PROGRAM F33_OuterPrinters_v2_Evo
VAR
	aSquareWave		 		: ARRAY[1..2] OF  FB_SquareWave;
	aOuterCodeGenerator 		: ARRAY[1..2] OF  FB_CODE_OuterCodeGenerator;
	aSelectCommand	 		: ARRAY[1..2] OF  FB_PRINTER_SelectCommand;

	aLabelPrintCtrl				: ARRAY[1..2] OF  RS;
	aLabelApplyCtrl			: ARRAY[1..2] OF  RS;

	tonLoweratorAtConstSpeed	: TON;
	rsInhibitLabbeller1Apply		: RS	;
	rsInhibitLabbeller2Apply		: RS	;

	fbDebugCNT				: FB_DEBUG_CounterArray;
	aCNTDebug				: ARRAY [1..10] OF UDINT;
	bResetCNT				: BOOL;
	bEnableResendCommand		: BOOL;
	rtEncoder	: R_TRIG;
END_VAR
VAR // added by the converter: edge detectors and wires of the graphical bodies
    _w1, _w2, _w3 : BOOL;
    _w4, _w5, _w6 : ANY;
END_VAR

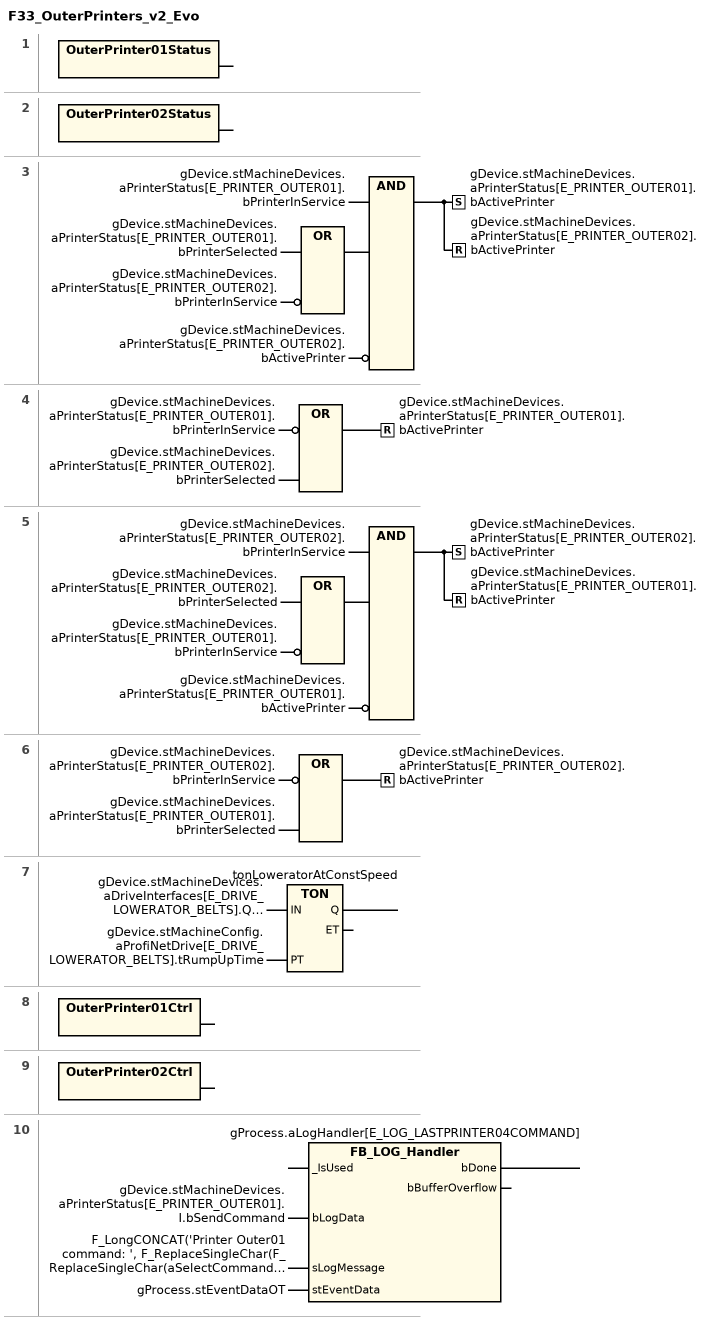
// NETWORK 1
OuterPrinter01Status();

// NETWORK 2
OuterPrinter02Status();

// NETWORK 3
_w1 := gDevice.stMachineDevices.aPrinterStatus[E_PRINTER_OUTER01].bPrinterInService AND (gDevice.stMachineDevices.aPrinterStatus[E_PRINTER_OUTER01].bPrinterSelected OR NOT gDevice.stMachineDevices.aPrinterStatus[E_PRINTER_OUTER02].bPrinterInService) AND NOT gDevice.stMachineDevices.aPrinterStatus[E_PRINTER_OUTER02].bActivePrinter;
gDevice.stMachineDevices.aPrinterStatus[E_PRINTER_OUTER01].bActivePrinter S= _w1;
gDevice.stMachineDevices.aPrinterStatus[E_PRINTER_OUTER02].bActivePrinter R= _w1;

// NETWORK 4
gDevice.stMachineDevices.aPrinterStatus[E_PRINTER_OUTER01].bActivePrinter R= NOT gDevice.stMachineDevices.aPrinterStatus[E_PRINTER_OUTER01].bPrinterInService OR gDevice.stMachineDevices.aPrinterStatus[E_PRINTER_OUTER02].bPrinterSelected;

// NETWORK 5
_w2 := gDevice.stMachineDevices.aPrinterStatus[E_PRINTER_OUTER02].bPrinterInService AND (gDevice.stMachineDevices.aPrinterStatus[E_PRINTER_OUTER02].bPrinterSelected OR NOT gDevice.stMachineDevices.aPrinterStatus[E_PRINTER_OUTER01].bPrinterInService) AND NOT gDevice.stMachineDevices.aPrinterStatus[E_PRINTER_OUTER01].bActivePrinter;
gDevice.stMachineDevices.aPrinterStatus[E_PRINTER_OUTER02].bActivePrinter S= _w2;
gDevice.stMachineDevices.aPrinterStatus[E_PRINTER_OUTER01].bActivePrinter R= _w2;

// NETWORK 6
gDevice.stMachineDevices.aPrinterStatus[E_PRINTER_OUTER02].bActivePrinter R= NOT gDevice.stMachineDevices.aPrinterStatus[E_PRINTER_OUTER02].bPrinterInService OR gDevice.stMachineDevices.aPrinterStatus[E_PRINTER_OUTER01].bPrinterSelected;

// NETWORK 7
tonLoweratorAtConstSpeed(IN := gDevice.stMachineDevices.aDriveInterfaces[E_DRIVE_LOWERATOR_BELTS].Q.xOperationEnable, PT := gDevice.stMachineConfig.aProfiNetDrive[E_DRIVE_LOWERATOR_BELTS].tRumpUpTime); // TON

// NETWORK 8
OuterPrinter01Ctrl();

// NETWORK 9
OuterPrinter02Ctrl();

// NETWORK 10
gProcess.aLogHandler[E_LOG_LASTPRINTER04COMMAND](
    bLogData := gDevice.stMachineDevices.aPrinterStatus[E_PRINTER_OUTER01].I.bSendCommand,
    sLogMessage := F_LongCONCAT('Printer Outer01 command: ', F_ReplaceSingleChar(F_ReplaceSingleChar(aSelectCommand[1].sPrintCommand, '$N', '_' ), '$R', '_')),
    stEventData := gProcess.stEventDataOT); // FB_LOG_Handler

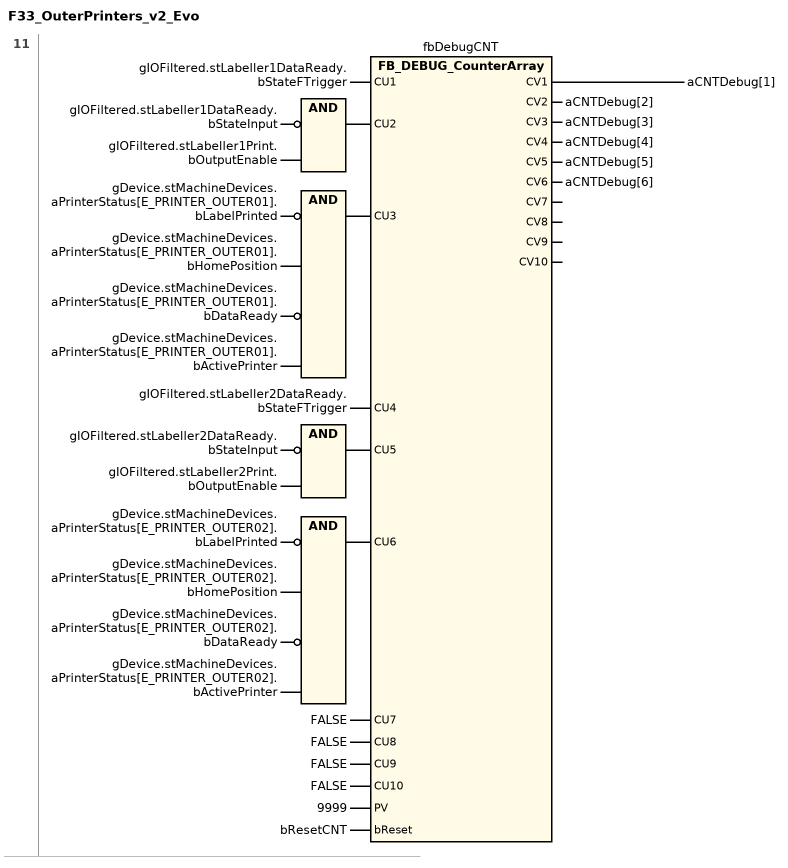
// NETWORK 11
fbDebugCNT(
    CU1 := gIOFiltered.stLabeller1DataReady.bStateFTrigger,
    CU2 := NOT gIOFiltered.stLabeller1DataReady.bStateInput AND gIOFiltered.stLabeller1Print.bOutputEnable,
    CU3 := NOT gDevice.stMachineDevices.aPrinterStatus[E_PRINTER_OUTER01].bLabelPrinted AND gDevice.stMachineDevices.aPrinterStatus[E_PRINTER_OUTER01].bHomePosition AND NOT gDevice.stMachineDevices.aPrinterStatus[E_PRINTER_OUTER01].bDataReady AND gDevice.stMachineDevices.aPrinterStatus[E_PRINTER_OUTER01].bActivePrinter,
    CU4 := gIOFiltered.stLabeller2DataReady.bStateFTrigger,
    CU5 := NOT gIOFiltered.stLabeller2DataReady.bStateInput AND gIOFiltered.stLabeller2Print.bOutputEnable,
    CU6 := NOT gDevice.stMachineDevices.aPrinterStatus[E_PRINTER_OUTER02].bLabelPrinted AND gDevice.stMachineDevices.aPrinterStatus[E_PRINTER_OUTER02].bHomePosition AND NOT gDevice.stMachineDevices.aPrinterStatus[E_PRINTER_OUTER02].bDataReady AND gDevice.stMachineDevices.aPrinterStatus[E_PRINTER_OUTER02].bActivePrinter,
    CU7 := FALSE,
    CU8 := FALSE,
    CU9 := FALSE,
    CU10 := FALSE,
    PV := 9999,
    bReset := bResetCNT,
    CV2 => aCNTDebug[2],
    CV3 => aCNTDebug[3],
    CV4 => aCNTDebug[4],
    CV5 => aCNTDebug[5],
    CV6 => aCNTDebug[6]); // FB_DEBUG_CounterArray
aCNTDebug[1] := fbDebugCNT.CV1;

ACTION OuterPrinter01Ctrl:
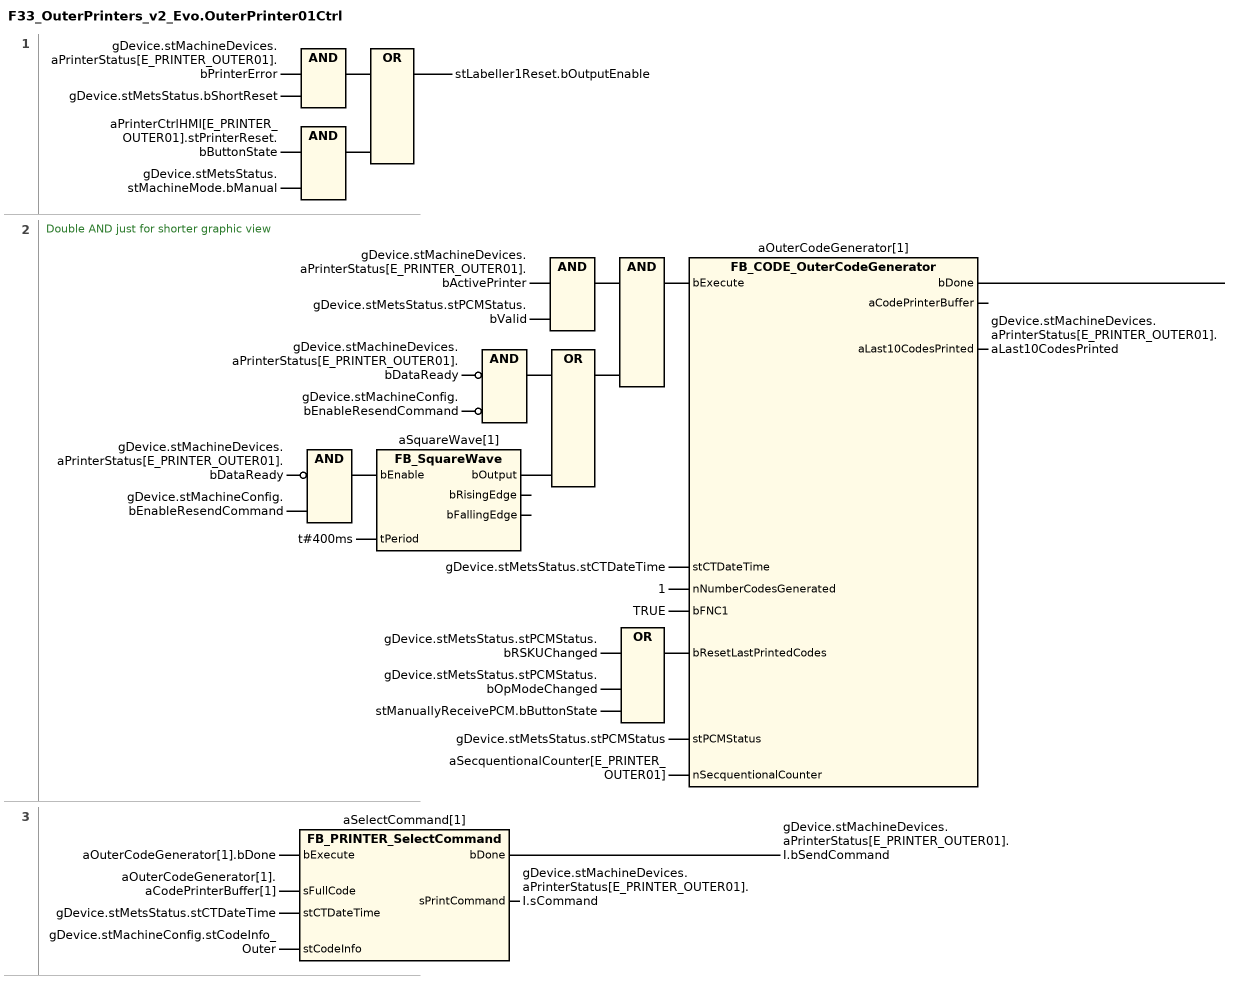
// NETWORK 1
stLabeller1Reset.bOutputEnable := gDevice.stMachineDevices.aPrinterStatus[E_PRINTER_OUTER01].bPrinterError AND gDevice.stMetsStatus.bShortReset OR aPrinterCtrlHMI[E_PRINTER_OUTER01].stPrinterReset.bButtonState AND gDevice.stMetsStatus.stMachineMode.bManual;

// NETWORK 2
// Double AND just for shorter graphic view
aSquareWave[1](bEnable := NOT gDevice.stMachineDevices.aPrinterStatus[E_PRINTER_OUTER01].bDataReady AND gDevice.stMachineConfig.bEnableResendCommand, tPeriod := t#400ms); // FB_SquareWave
aOuterCodeGenerator[1](
    bExecute := (gDevice.stMachineDevices.aPrinterStatus[E_PRINTER_OUTER01].bActivePrinter AND gDevice.stMetsStatus.stPCMStatus.bValid) AND (NOT gDevice.stMachineDevices.aPrinterStatus[E_PRINTER_OUTER01].bDataReady AND NOT gDevice.stMachineConfig.bEnableResendCommand OR aSquareWave[1].bOutput),
    stCTDateTime := gDevice.stMetsStatus.stCTDateTime,
    nNumberCodesGenerated := 1,
    bFNC1 := TRUE,
    bResetLastPrintedCodes := gDevice.stMetsStatus.stPCMStatus.bRSKUChanged OR gDevice.stMetsStatus.stPCMStatus.bOpModeChanged OR stManuallyReceivePCM.bButtonState,
    stPCMStatus := gDevice.stMetsStatus.stPCMStatus,
    nSecquentionalCounter := aSecquentionalCounter[E_PRINTER_OUTER01],
    aLast10CodesPrinted => gDevice.stMachineDevices.aPrinterStatus[E_PRINTER_OUTER01].aLast10CodesPrinted); // FB_CODE_OuterCodeGenerator

// NETWORK 3
aSelectCommand[1](
    bExecute := aOuterCodeGenerator[1].bDone,
    sFullCode := aOuterCodeGenerator[1].aCodePrinterBuffer[1],
    stCTDateTime := gDevice.stMetsStatus.stCTDateTime,
    stCodeInfo := gDevice.stMachineConfig.stCodeInfo_Outer,
    sPrintCommand => gDevice.stMachineDevices.aPrinterStatus[E_PRINTER_OUTER01].I.sCommand); // FB_PRINTER_SelectCommand
gDevice.stMachineDevices.aPrinterStatus[E_PRINTER_OUTER01].I.bSendCommand := aSelectCommand[1].bDone;

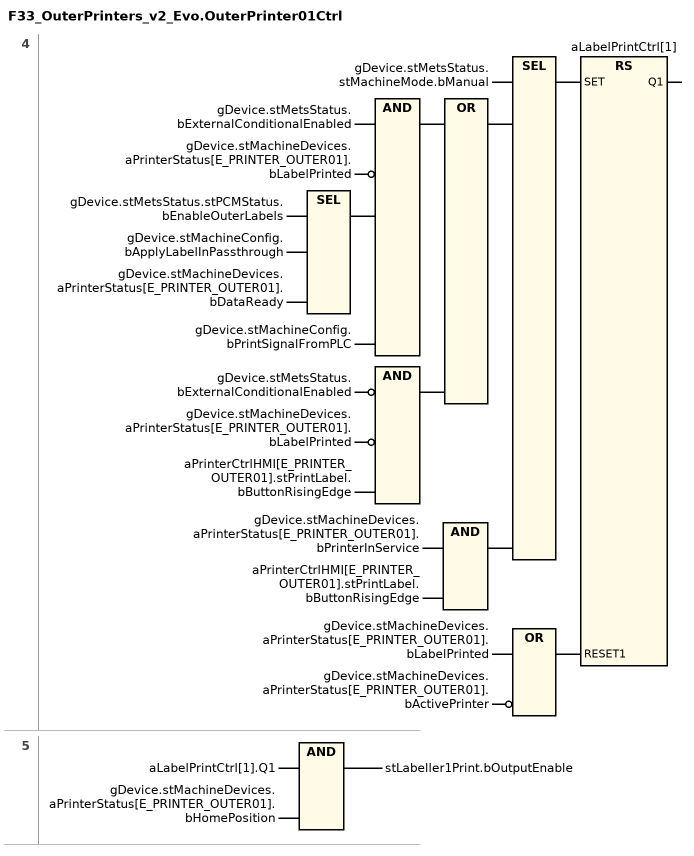
// NETWORK 4
aLabelPrintCtrl[1](SET := SEL(gDevice.stMetsStatus.stMachineMode.bManual, gDevice.stMetsStatus.bExternalConditionalEnabled AND NOT gDevice.stMachineDevices.aPrinterStatus[E_PRINTER_OUTER01].bLabelPrinted AND SEL(gDevice.stMetsStatus.stPCMStatus.bEnableOuterLabels, gDevice.stMachineConfig.bApplyLabelInPassthrough, gDevice.stMachineDevices.aPrinterStatus[E_PRINTER_OUTER01].bDataReady) AND gDevice.stMachineConfig.bPrintSignalFromPLC OR NOT gDevice.stMetsStatus.bExternalConditionalEnabled AND NOT gDevice.stMachineDevices.aPrinterStatus[E_PRINTER_OUTER01].bLabelPrinted AND aPrinterCtrlHMI[E_PRINTER_OUTER01].stPrintLabel.bButtonRisingEdge, gDevice.stMachineDevices.aPrinterStatus[E_PRINTER_OUTER01].bPrinterInService AND aPrinterCtrlHMI[E_PRINTER_OUTER01].stPrintLabel.bButtonRisingEdge), RESET1 := gDevice.stMachineDevices.aPrinterStatus[E_PRINTER_OUTER01].bLabelPrinted OR NOT gDevice.stMachineDevices.aPrinterStatus[E_PRINTER_OUTER01].bActivePrinter); // RS

// NETWORK 5
stLabeller1Print.bOutputEnable := aLabelPrintCtrl[1].Q1 AND gDevice.stMachineDevices.aPrinterStatus[E_PRINTER_OUTER01].bHomePosition;

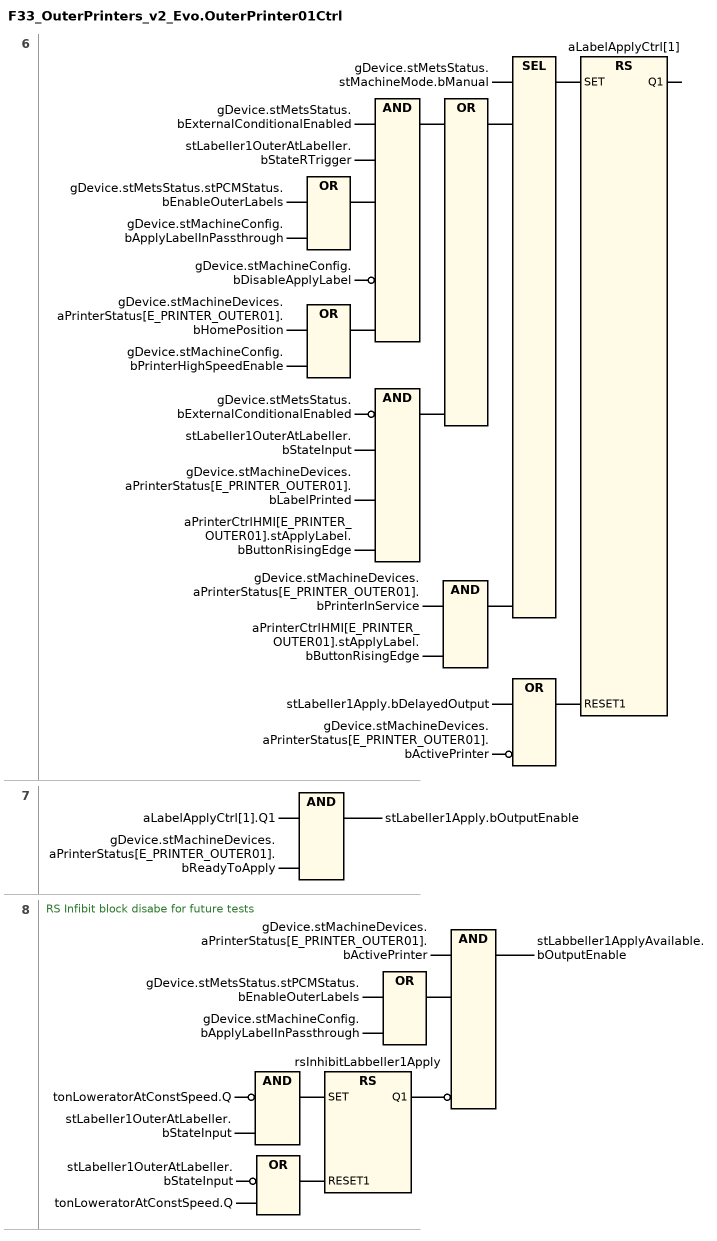
// NETWORK 6
aLabelApplyCtrl[1](SET := SEL(gDevice.stMetsStatus.stMachineMode.bManual, gDevice.stMetsStatus.bExternalConditionalEnabled AND stLabeller1OuterAtLabeller.bStateRTrigger AND (gDevice.stMetsStatus.stPCMStatus.bEnableOuterLabels OR gDevice.stMachineConfig.bApplyLabelInPassthrough) AND NOT gDevice.stMachineConfig.bDisableApplyLabel AND (gDevice.stMachineDevices.aPrinterStatus[E_PRINTER_OUTER01].bHomePosition OR gDevice.stMachineConfig.bPrinterHighSpeedEnable) OR NOT gDevice.stMetsStatus.bExternalConditionalEnabled AND stLabeller1OuterAtLabeller.bStateInput AND gDevice.stMachineDevices.aPrinterStatus[E_PRINTER_OUTER01].bLabelPrinted AND aPrinterCtrlHMI[E_PRINTER_OUTER01].stApplyLabel.bButtonRisingEdge, gDevice.stMachineDevices.aPrinterStatus[E_PRINTER_OUTER01].bPrinterInService AND aPrinterCtrlHMI[E_PRINTER_OUTER01].stApplyLabel.bButtonRisingEdge), RESET1 := stLabeller1Apply.bDelayedOutput OR NOT gDevice.stMachineDevices.aPrinterStatus[E_PRINTER_OUTER01].bActivePrinter); // RS

// NETWORK 7
stLabeller1Apply.bOutputEnable := aLabelApplyCtrl[1].Q1 AND gDevice.stMachineDevices.aPrinterStatus[E_PRINTER_OUTER01].bReadyToApply;

// NETWORK 8
// RS Infibit block disabe for future tests
rsInhibitLabbeller1Apply(SET := NOT tonLoweratorAtConstSpeed.Q AND stLabeller1OuterAtLabeller.bStateInput, RESET1 := NOT stLabeller1OuterAtLabeller.bStateInput OR tonLoweratorAtConstSpeed.Q); // RS
stLabbeller1ApplyAvailable.bOutputEnable := gDevice.stMachineDevices.aPrinterStatus[E_PRINTER_OUTER01].bActivePrinter AND (gDevice.stMetsStatus.stPCMStatus.bEnableOuterLabels OR gDevice.stMachineConfig.bApplyLabelInPassthrough) AND NOT rsInhibitLabbeller1Apply.Q1;
END_ACTION

ACTION OuterPrinter01Status:
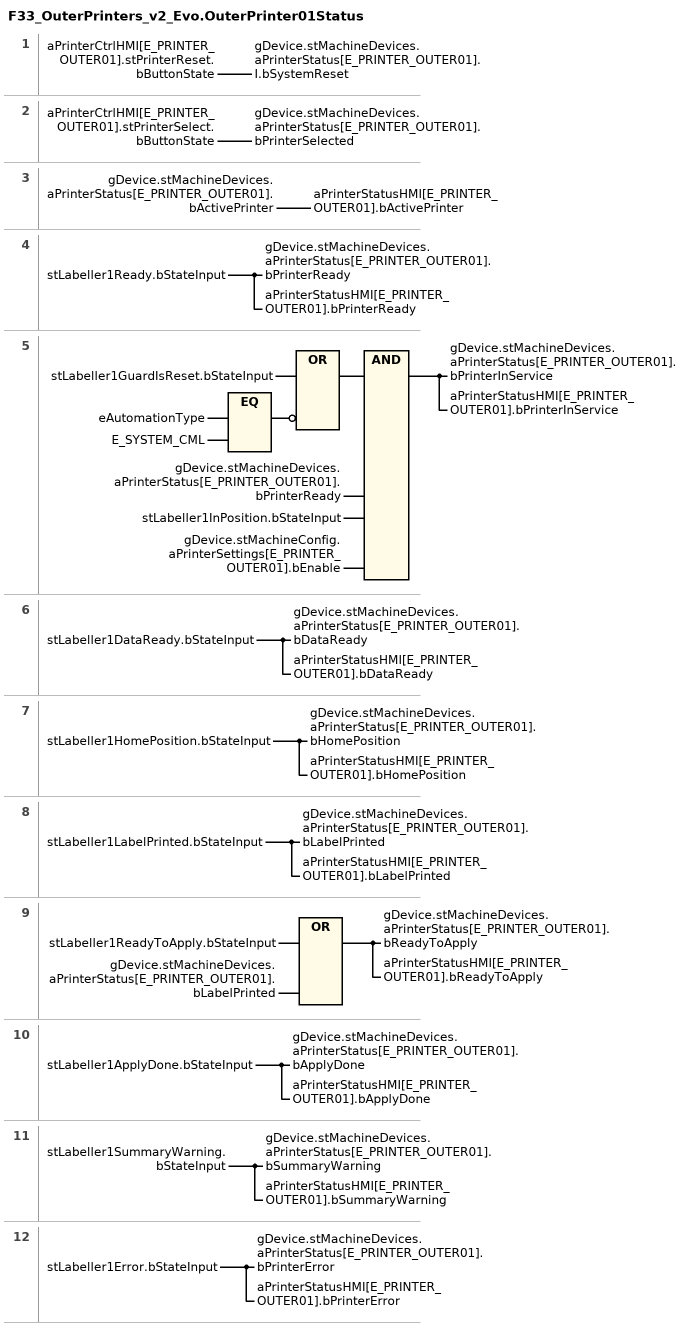
// NETWORK 1
gDevice.stMachineDevices.aPrinterStatus[E_PRINTER_OUTER01].I.bSystemReset := aPrinterCtrlHMI[E_PRINTER_OUTER01].stPrinterReset.bButtonState;

// NETWORK 2
gDevice.stMachineDevices.aPrinterStatus[E_PRINTER_OUTER01].bPrinterSelected := aPrinterCtrlHMI[E_PRINTER_OUTER01].stPrinterSelect.bButtonState;

// NETWORK 3
aPrinterStatusHMI[E_PRINTER_OUTER01].bActivePrinter := gDevice.stMachineDevices.aPrinterStatus[E_PRINTER_OUTER01].bActivePrinter;

// NETWORK 4
gDevice.stMachineDevices.aPrinterStatus[E_PRINTER_OUTER01].bPrinterReady := stLabeller1Ready.bStateInput;
aPrinterStatusHMI[E_PRINTER_OUTER01].bPrinterReady := stLabeller1Ready.bStateInput;

// NETWORK 5
_w3 := (stLabeller1GuardIsReset.bStateInput OR NOT (eAutomationType = E_SYSTEM_CML)) AND gDevice.stMachineDevices.aPrinterStatus[E_PRINTER_OUTER01].bPrinterReady AND stLabeller1InPosition.bStateInput AND gDevice.stMachineConfig.aPrinterSettings[E_PRINTER_OUTER01].bEnable;
gDevice.stMachineDevices.aPrinterStatus[E_PRINTER_OUTER01].bPrinterInService := _w3;
aPrinterStatusHMI[E_PRINTER_OUTER01].bPrinterInService := _w3;

// NETWORK 6
gDevice.stMachineDevices.aPrinterStatus[E_PRINTER_OUTER01].bDataReady := stLabeller1DataReady.bStateInput;
aPrinterStatusHMI[E_PRINTER_OUTER01].bDataReady := stLabeller1DataReady.bStateInput;

// NETWORK 7
gDevice.stMachineDevices.aPrinterStatus[E_PRINTER_OUTER01].bHomePosition := stLabeller1HomePosition.bStateInput;
aPrinterStatusHMI[E_PRINTER_OUTER01].bHomePosition := stLabeller1HomePosition.bStateInput;

// NETWORK 8
gDevice.stMachineDevices.aPrinterStatus[E_PRINTER_OUTER01].bLabelPrinted := stLabeller1LabelPrinted.bStateInput;
aPrinterStatusHMI[E_PRINTER_OUTER01].bLabelPrinted := stLabeller1LabelPrinted.bStateInput;

// NETWORK 9
_w4 := stLabeller1ReadyToApply.bStateInput OR gDevice.stMachineDevices.aPrinterStatus[E_PRINTER_OUTER01].bLabelPrinted;
gDevice.stMachineDevices.aPrinterStatus[E_PRINTER_OUTER01].bReadyToApply := _w4;
aPrinterStatusHMI[E_PRINTER_OUTER01].bReadyToApply := _w4;

// NETWORK 10
gDevice.stMachineDevices.aPrinterStatus[E_PRINTER_OUTER01].bApplyDone := stLabeller1ApplyDone.bStateInput;
aPrinterStatusHMI[E_PRINTER_OUTER01].bApplyDone := stLabeller1ApplyDone.bStateInput;

// NETWORK 11
gDevice.stMachineDevices.aPrinterStatus[E_PRINTER_OUTER01].bSummaryWarning := stLabeller1SummaryWarning.bStateInput;
aPrinterStatusHMI[E_PRINTER_OUTER01].bSummaryWarning := stLabeller1SummaryWarning.bStateInput;

// NETWORK 12
gDevice.stMachineDevices.aPrinterStatus[E_PRINTER_OUTER01].bPrinterError := stLabeller1Error.bStateInput;
aPrinterStatusHMI[E_PRINTER_OUTER01].bPrinterError := stLabeller1Error.bStateInput;
END_ACTION

ACTION OuterPrinter02Ctrl:
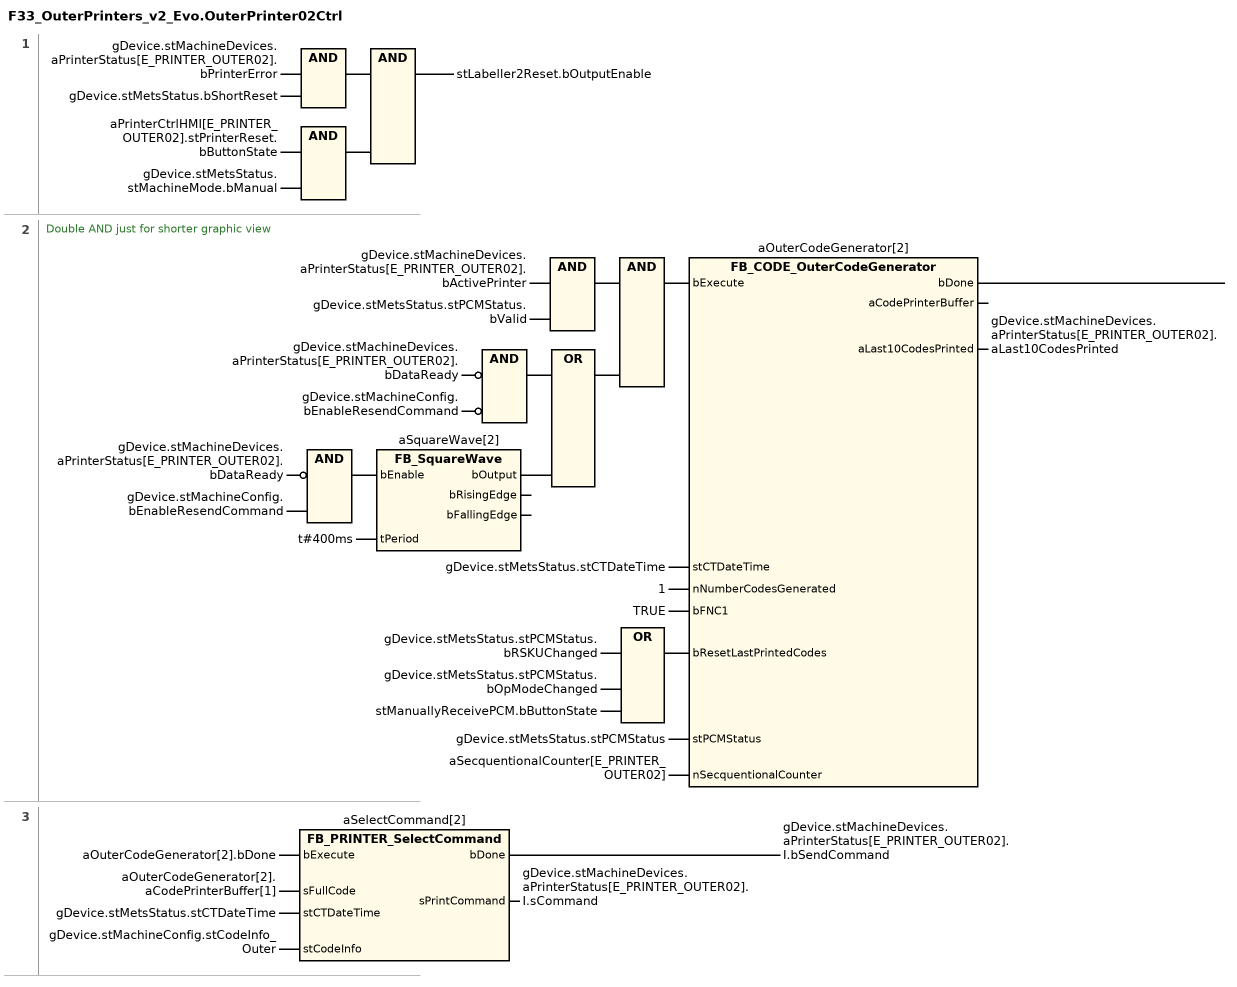
// NETWORK 1
stLabeller2Reset.bOutputEnable := (gDevice.stMachineDevices.aPrinterStatus[E_PRINTER_OUTER02].bPrinterError AND gDevice.stMetsStatus.bShortReset) AND (aPrinterCtrlHMI[E_PRINTER_OUTER02].stPrinterReset.bButtonState AND gDevice.stMetsStatus.stMachineMode.bManual);

// NETWORK 2
// Double AND just for shorter graphic view
aSquareWave[2](bEnable := NOT gDevice.stMachineDevices.aPrinterStatus[E_PRINTER_OUTER02].bDataReady AND gDevice.stMachineConfig.bEnableResendCommand, tPeriod := t#400ms); // FB_SquareWave
aOuterCodeGenerator[2](
    bExecute := (gDevice.stMachineDevices.aPrinterStatus[E_PRINTER_OUTER02].bActivePrinter AND gDevice.stMetsStatus.stPCMStatus.bValid) AND (NOT gDevice.stMachineDevices.aPrinterStatus[E_PRINTER_OUTER02].bDataReady AND NOT gDevice.stMachineConfig.bEnableResendCommand OR aSquareWave[2].bOutput),
    stCTDateTime := gDevice.stMetsStatus.stCTDateTime,
    nNumberCodesGenerated := 1,
    bFNC1 := TRUE,
    bResetLastPrintedCodes := gDevice.stMetsStatus.stPCMStatus.bRSKUChanged OR gDevice.stMetsStatus.stPCMStatus.bOpModeChanged OR stManuallyReceivePCM.bButtonState,
    stPCMStatus := gDevice.stMetsStatus.stPCMStatus,
    nSecquentionalCounter := aSecquentionalCounter[E_PRINTER_OUTER02],
    aLast10CodesPrinted => gDevice.stMachineDevices.aPrinterStatus[E_PRINTER_OUTER02].aLast10CodesPrinted); // FB_CODE_OuterCodeGenerator

// NETWORK 3
aSelectCommand[2](
    bExecute := aOuterCodeGenerator[2].bDone,
    sFullCode := aOuterCodeGenerator[2].aCodePrinterBuffer[1],
    stCTDateTime := gDevice.stMetsStatus.stCTDateTime,
    stCodeInfo := gDevice.stMachineConfig.stCodeInfo_Outer,
    sPrintCommand => gDevice.stMachineDevices.aPrinterStatus[E_PRINTER_OUTER02].I.sCommand); // FB_PRINTER_SelectCommand
gDevice.stMachineDevices.aPrinterStatus[E_PRINTER_OUTER02].I.bSendCommand := aSelectCommand[2].bDone;

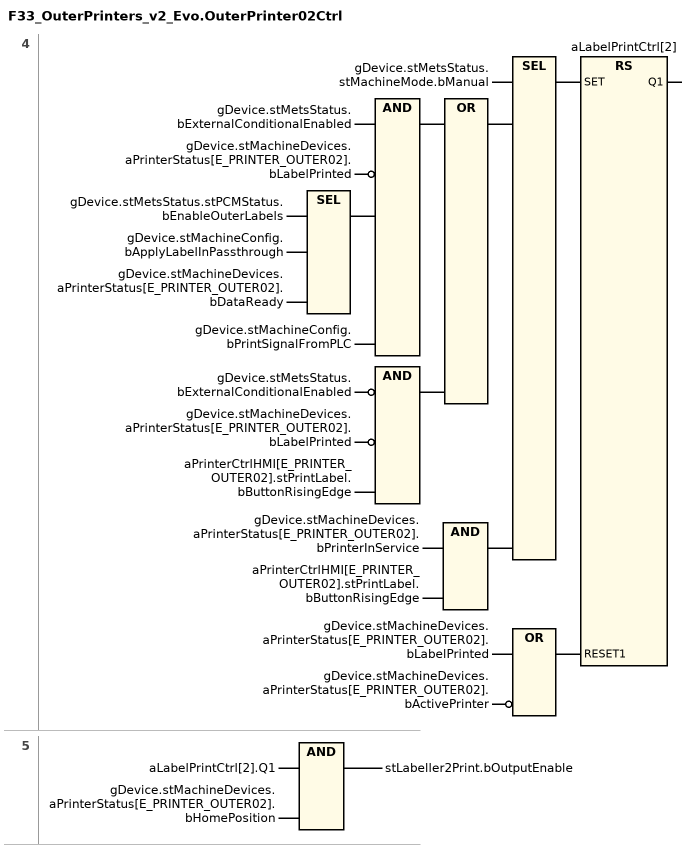
// NETWORK 4
aLabelPrintCtrl[2](SET := SEL(gDevice.stMetsStatus.stMachineMode.bManual, gDevice.stMetsStatus.bExternalConditionalEnabled AND NOT gDevice.stMachineDevices.aPrinterStatus[E_PRINTER_OUTER02].bLabelPrinted AND SEL(gDevice.stMetsStatus.stPCMStatus.bEnableOuterLabels, gDevice.stMachineConfig.bApplyLabelInPassthrough, gDevice.stMachineDevices.aPrinterStatus[E_PRINTER_OUTER02].bDataReady) AND gDevice.stMachineConfig.bPrintSignalFromPLC OR NOT gDevice.stMetsStatus.bExternalConditionalEnabled AND NOT gDevice.stMachineDevices.aPrinterStatus[E_PRINTER_OUTER02].bLabelPrinted AND aPrinterCtrlHMI[E_PRINTER_OUTER02].stPrintLabel.bButtonRisingEdge, gDevice.stMachineDevices.aPrinterStatus[E_PRINTER_OUTER02].bPrinterInService AND aPrinterCtrlHMI[E_PRINTER_OUTER02].stPrintLabel.bButtonRisingEdge), RESET1 := gDevice.stMachineDevices.aPrinterStatus[E_PRINTER_OUTER02].bLabelPrinted OR NOT gDevice.stMachineDevices.aPrinterStatus[E_PRINTER_OUTER02].bActivePrinter); // RS

// NETWORK 5
stLabeller2Print.bOutputEnable := aLabelPrintCtrl[2].Q1 AND gDevice.stMachineDevices.aPrinterStatus[E_PRINTER_OUTER02].bHomePosition;

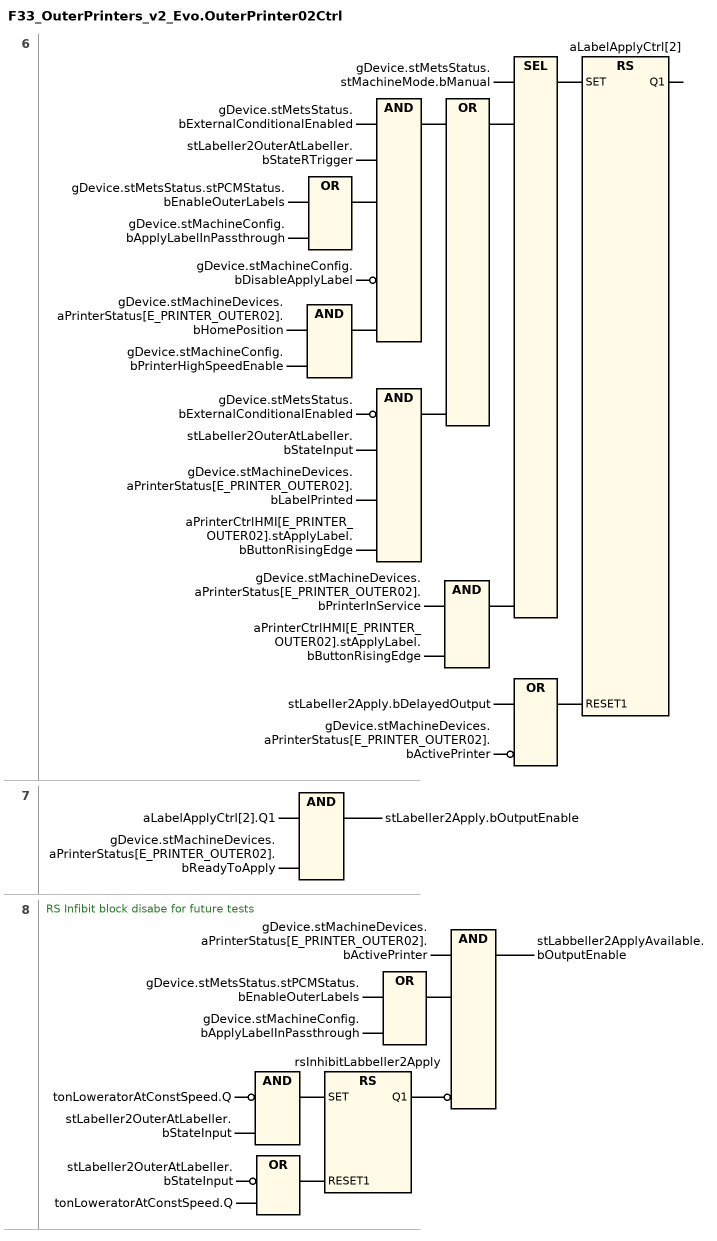
// NETWORK 6
aLabelApplyCtrl[2](SET := SEL(gDevice.stMetsStatus.stMachineMode.bManual, gDevice.stMetsStatus.bExternalConditionalEnabled AND stLabeller2OuterAtLabeller.bStateRTrigger AND (gDevice.stMetsStatus.stPCMStatus.bEnableOuterLabels OR gDevice.stMachineConfig.bApplyLabelInPassthrough) AND NOT gDevice.stMachineConfig.bDisableApplyLabel AND (gDevice.stMachineDevices.aPrinterStatus[E_PRINTER_OUTER02].bHomePosition AND gDevice.stMachineConfig.bPrinterHighSpeedEnable) OR NOT gDevice.stMetsStatus.bExternalConditionalEnabled AND stLabeller2OuterAtLabeller.bStateInput AND gDevice.stMachineDevices.aPrinterStatus[E_PRINTER_OUTER02].bLabelPrinted AND aPrinterCtrlHMI[E_PRINTER_OUTER02].stApplyLabel.bButtonRisingEdge, gDevice.stMachineDevices.aPrinterStatus[E_PRINTER_OUTER02].bPrinterInService AND aPrinterCtrlHMI[E_PRINTER_OUTER02].stApplyLabel.bButtonRisingEdge), RESET1 := stLabeller2Apply.bDelayedOutput OR NOT gDevice.stMachineDevices.aPrinterStatus[E_PRINTER_OUTER02].bActivePrinter); // RS

// NETWORK 7
stLabeller2Apply.bOutputEnable := aLabelApplyCtrl[2].Q1 AND gDevice.stMachineDevices.aPrinterStatus[E_PRINTER_OUTER02].bReadyToApply;

// NETWORK 8
// RS Infibit block disabe for future tests
rsInhibitLabbeller2Apply(SET := NOT tonLoweratorAtConstSpeed.Q AND stLabeller2OuterAtLabeller.bStateInput, RESET1 := NOT stLabeller2OuterAtLabeller.bStateInput OR tonLoweratorAtConstSpeed.Q); // RS
stLabbeller2ApplyAvailable.bOutputEnable := gDevice.stMachineDevices.aPrinterStatus[E_PRINTER_OUTER02].bActivePrinter AND (gDevice.stMetsStatus.stPCMStatus.bEnableOuterLabels OR gDevice.stMachineConfig.bApplyLabelInPassthrough) AND NOT rsInhibitLabbeller2Apply.Q1;
END_ACTION

ACTION OuterPrinter02Status:
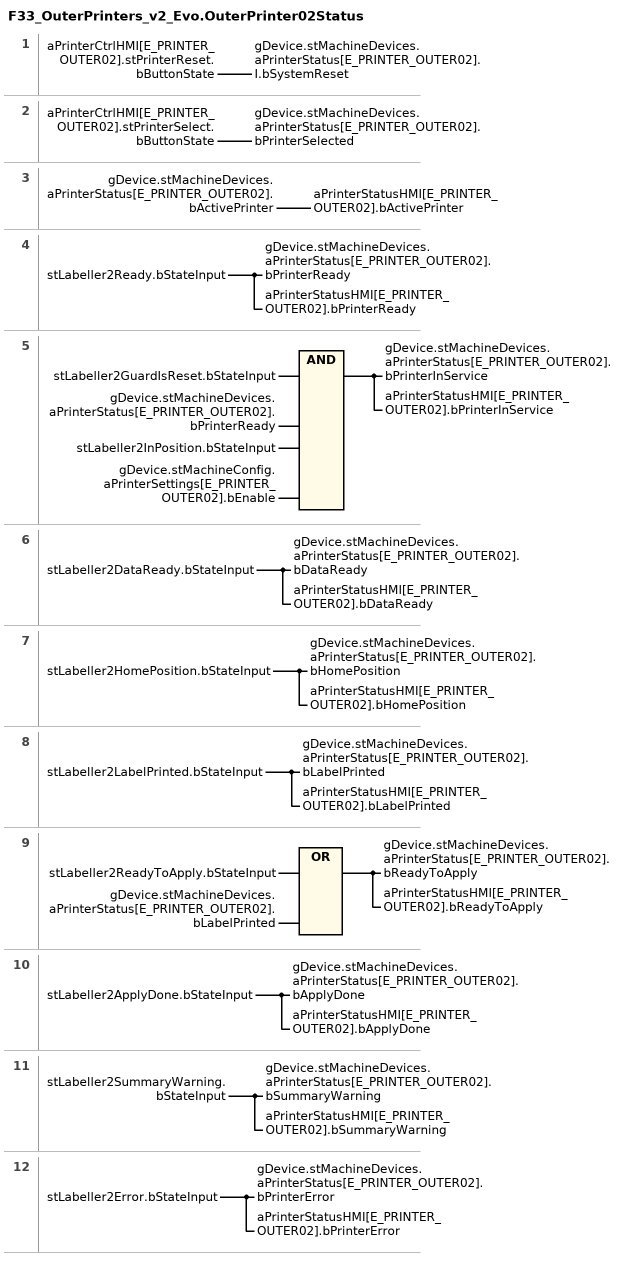
// NETWORK 1
gDevice.stMachineDevices.aPrinterStatus[E_PRINTER_OUTER02].I.bSystemReset := aPrinterCtrlHMI[E_PRINTER_OUTER02].stPrinterReset.bButtonState;

// NETWORK 2
gDevice.stMachineDevices.aPrinterStatus[E_PRINTER_OUTER02].bPrinterSelected := aPrinterCtrlHMI[E_PRINTER_OUTER02].stPrinterSelect.bButtonState;

// NETWORK 3
aPrinterStatusHMI[E_PRINTER_OUTER02].bActivePrinter := gDevice.stMachineDevices.aPrinterStatus[E_PRINTER_OUTER02].bActivePrinter;

// NETWORK 4
gDevice.stMachineDevices.aPrinterStatus[E_PRINTER_OUTER02].bPrinterReady := stLabeller2Ready.bStateInput;
aPrinterStatusHMI[E_PRINTER_OUTER02].bPrinterReady := stLabeller2Ready.bStateInput;

// NETWORK 5
_w5 := stLabeller2GuardIsReset.bStateInput AND gDevice.stMachineDevices.aPrinterStatus[E_PRINTER_OUTER02].bPrinterReady AND stLabeller2InPosition.bStateInput AND gDevice.stMachineConfig.aPrinterSettings[E_PRINTER_OUTER02].bEnable;
gDevice.stMachineDevices.aPrinterStatus[E_PRINTER_OUTER02].bPrinterInService := _w5;
aPrinterStatusHMI[E_PRINTER_OUTER02].bPrinterInService := _w5;

// NETWORK 6
gDevice.stMachineDevices.aPrinterStatus[E_PRINTER_OUTER02].bDataReady := stLabeller2DataReady.bStateInput;
aPrinterStatusHMI[E_PRINTER_OUTER02].bDataReady := stLabeller2DataReady.bStateInput;

// NETWORK 7
gDevice.stMachineDevices.aPrinterStatus[E_PRINTER_OUTER02].bHomePosition := stLabeller2HomePosition.bStateInput;
aPrinterStatusHMI[E_PRINTER_OUTER02].bHomePosition := stLabeller2HomePosition.bStateInput;

// NETWORK 8
gDevice.stMachineDevices.aPrinterStatus[E_PRINTER_OUTER02].bLabelPrinted := stLabeller2LabelPrinted.bStateInput;
aPrinterStatusHMI[E_PRINTER_OUTER02].bLabelPrinted := stLabeller2LabelPrinted.bStateInput;

// NETWORK 9
_w6 := stLabeller2ReadyToApply.bStateInput OR gDevice.stMachineDevices.aPrinterStatus[E_PRINTER_OUTER02].bLabelPrinted;
gDevice.stMachineDevices.aPrinterStatus[E_PRINTER_OUTER02].bReadyToApply := _w6;
aPrinterStatusHMI[E_PRINTER_OUTER02].bReadyToApply := _w6;

// NETWORK 10
gDevice.stMachineDevices.aPrinterStatus[E_PRINTER_OUTER02].bApplyDone := stLabeller2ApplyDone.bStateInput;
aPrinterStatusHMI[E_PRINTER_OUTER02].bApplyDone := stLabeller2ApplyDone.bStateInput;

// NETWORK 11
gDevice.stMachineDevices.aPrinterStatus[E_PRINTER_OUTER02].bSummaryWarning := stLabeller2SummaryWarning.bStateInput;
aPrinterStatusHMI[E_PRINTER_OUTER02].bSummaryWarning := stLabeller2SummaryWarning.bStateInput;

// NETWORK 12
gDevice.stMachineDevices.aPrinterStatus[E_PRINTER_OUTER02].bPrinterError := stLabeller2Error.bStateInput;
aPrinterStatusHMI[E_PRINTER_OUTER02].bPrinterError := stLabeller2Error.bStateInput;
END_ACTION

END_PROGRAM

(* stored: Version 1.1.0.1
   POU F33_OuterPrinters_v2_Evo: Id {f0037de4-57c9-48c3-b72c-de81e2c0d60b}, SpecialFunc None
   Action OuterPrinter01Ctrl: Id {3914b2ef-d6db-48ac-bc80-f076a72e2194}
   Action OuterPrinter01Status: Id {b2b77f8a-4f3c-4042-a8c5-671c1d37948e}
   Action OuterPrinter02Ctrl: Id {2c47a344-ac70-4596-b683-54381d2f5192}
   Action OuterPrinter02Status: Id {a3f6eb7d-695d-4b7d-841a-3f8c22097dad} *)
